Fanuc KAREL source: kt00340.KL

PROGRAM KT00340
%NOLOCKGROUP
VAR
Y1 : ARRAY[2] OF BYTE
R2:REAL
OUT:BOOLEAN
BEGIN
Y1[1]=2
R2=3.0
OUT=((Y1[1])<R2)
END KT00340
